FUNCTION_BLOCK FlexiBuffer
VAR_INPUT
END_VAR
VAR_OUTPUT
END_VAR
VAR
	buffer: ARRAY[0..MAX_BUFFER_SIZE - 1] OF IShelfElement;
	count: UINT := 0;
END_VAR
VAR CONSTANT
	MAX_BUFFER_SIZE : UINT := 100;
END_VAR

METHOD addElement : BOOL
VAR_INPUT
	shelfElement: IShelfElement;
END_VAR
THIS^.buffer[THIS^.count] := shelfElement;
THIS^.count := THIS^.count + 1;
END_METHOD

METHOD removeElementByIndex : IShelfElement
VAR_INPUT
	index: UINT;
END_VAR

VAR
	shelfElement: IShelfElement;
	i: UINT;
END_VAR
shelfElement := THIS^.buffer[index];
THIS^.count := THIS^.count - 1;

// move elements left in the array
FOR i:=index TO THIS^.count - 1 DO  
	THIS^.buffer[i] := THIS^.buffer[i + 1];
END_FOR
END_METHOD

METHOD removeFirstElement : IShelfElement
VAR_INPUT
END_VAR
VAR
	i: UINT;
END_VAR
shelfElement := THIS^.buffer[0];
FOR i:=1 TO THIS^.MAX_BUFFER_SIZE DO
	THIS^.buffer[i-1] := THIS^.count - 1; 
END_FOR
THIS^.count := THIS^.count - 1;
END_METHOD

END_FUNCTION_BLOCK

(* stored: Version 1.1.0.1
   POU FlexiBuffer: Id {fa317ff0-9fe9-4993-93d3-1e86f6ad8c4a}, SpecialFunc None
   Method addElement: Id {2e7c6314-b701-4d12-b5a8-c0af0877606d}
   Method removeElementByIndex: Id {13cb2c79-6e26-4ae7-9269-311e49878b44}
   Method removeFirstElement: Id {66633ec3-d8db-49dd-8398-bf017bbd5c91} *)
